// TIA Portal project "Servo With PLC" (V18)

(* hardware
DEVICE "S7-1200 station_1"  S7-1200 Station
   slot 0: "Rack_0"  S7-1200 Rack  Rack  V1.0
   slot 1: "PLC_1"  CPU 1215C DC/DC/DC  6ES7 215-1AG40-0XB0  V4.6
*)

// ===== PLC "PLC_1"  CPU 1215C DC/DC/DC =====

VAR_GLOBAL   // PLC tag table "Default tag table"
   "Servo Control_Pulse" AT %Q0.0 : Bool;
   "Servo Control_Direction" AT %Q0.1 : Bool;
   "Servo Control_DriveEnable" AT %Q0.2 : Bool;
   "Tag_1" AT %M0.0 : Bool;
   "Tag_2" AT %M0.1 : Bool;
   "Tag_3" AT %M0.2 : Bool;
   "Tag_4" AT %M0.3 : Bool;
   "Velocity for JOG" AT %MD10 : Real;
   "Tag_5" AT %M0.4 : Bool;
   "Tag_6" AT %MD14 : Real;
   "Tag_7" AT %MD18 : Real;
   "TotalTime (S)" AT %MD22 : Real;
   "tagg" AT %MD26 : Real;
   "Final Distance (mm)" AT %MD24 : Real;
   "final distance (mm)(1)" AT %MD30 : Real;
   "Tag_8" AT %M0.5 : Bool;
   "Tag_9" AT %M0.6 : Bool;
   "Tag_10" AT %MD34 : Real;
   "Tag_11" AT %MD38 : Real;
END_VAR

DATA_BLOCK "Servo Control"   // DB1, Motion_DB
{ S7_Optimized_Access := 'TRUE' }
AUTHOR : SIMATIC
FAMILY : BasicMC
NAME : TO_PosAx
VERSION : 8.0
// stored: InstanceOfName TO_PositioningAxis
"TO_PositioningAxis"
BEGIN
   // Axis.EnableOutput_AddressCU = %Q0.2
   // Axis.LengthUnit.LastDistance = -1
   // Axis.OnlinePtoModeCU = 16#0000_0002
   // Axis.DirectionOutputEnabledCU = TRUE
   // Axis.SelectedChannel2EnumCU = %Q0.1
   // Axis.SelectedChannel1EnumCU = %Q0.0
   // Pulse.MinDeltaDeltaFrequencyCU = 0.004
   // Pulse.MaxDeltaDeltaFrequencyCU = 1.0E+10
   // Pulse.MinDeltaFrequencyCU = 0.005
   // Pulse.MaxDeltaFrequencyCU = 9.5E+9
   // Pulse.MinFrequencyCU = 1.0
   // Pulse.MaxFrequencyCU = 100000.0
   // Pulse.OutputSourceCU = 16#0000_0000
   // Axis.SelectPTO = 0
END_DATA_BLOCK

ORGANIZATION_BLOCK "Main"   // OB1, LAD, ProgramCycle
TITLE = "Main Program Sweep (Cycle)"
{ S7_Optimized_Access := 'TRUE' }
VERSION : 0.1
   VAR_INPUT
      Initial_Call : Bool;   // Initial call of this OB
      Remanence : Bool;   // =True, if remanent data are available
   END_VAR
BEGIN

REGION Network 1
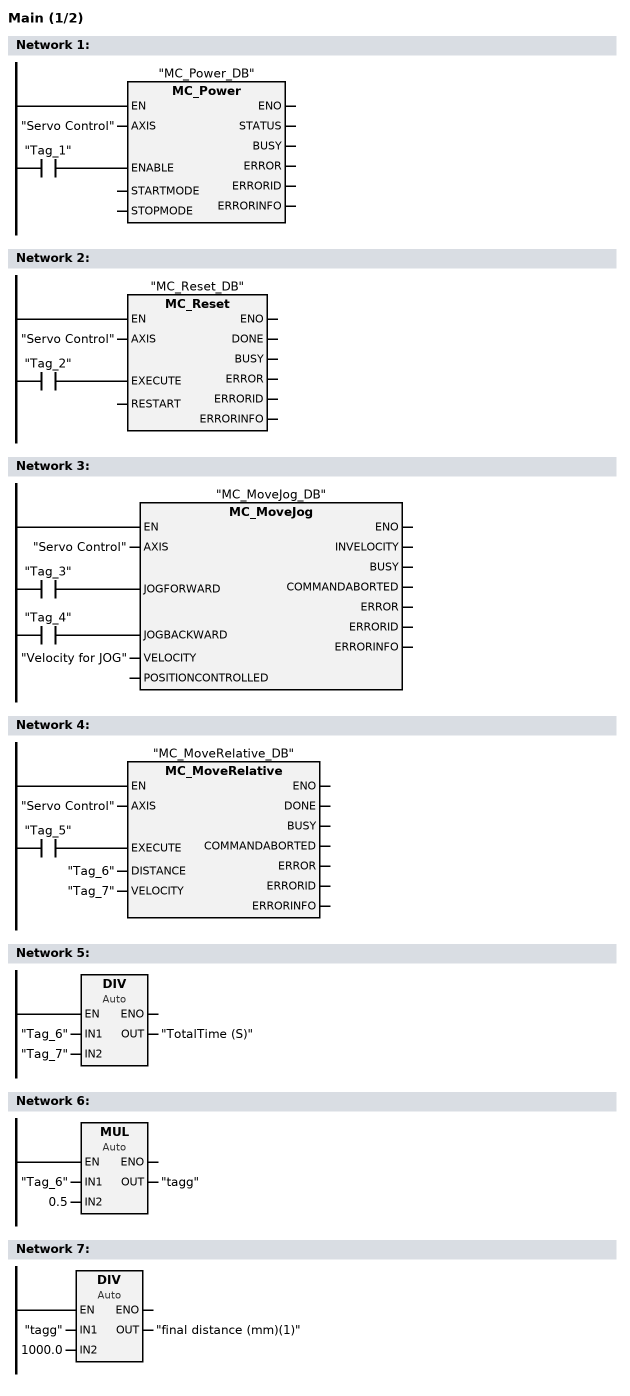
   "MC_Power_DB"(Axis := "Servo Control", Enable := "Tag_1");   // MC_Power
END_REGION

REGION Network 2
   "MC_Reset_DB"(Axis := "Servo Control", Execute := "Tag_2");   // MC_Reset
END_REGION

REGION Network 3
   "MC_MoveJog_DB"(Axis := "Servo Control",   // MC_MoveJog
                   JogForward := "Tag_3",
                   JogBackward := "Tag_4",
                   Velocity := "Velocity for JOG");
END_REGION

REGION Network 4
   "MC_MoveRelative_DB"(Axis := "Servo Control", Execute := "Tag_5", Distance := "Tag_6", Velocity := "Tag_7");   // MC_MoveRelative
END_REGION

REGION Network 5
   RUNG wire#powerrail
      Div(in1 := "Tag_6", in2 := "Tag_7", out => "TotalTime (S)")
   END_RUNG
   // the same network as SCL:
   "TotalTime (S)" := "Tag_6" / "Tag_7";
END_REGION

REGION Network 6
   RUNG wire#powerrail
      Mul(in1 := "Tag_6", in2 := 0.5, out => "tagg")
   END_RUNG
   // the same network as SCL:
   "tagg" := "Tag_6" * 0.5;
END_REGION

REGION Network 7
   RUNG wire#powerrail
      Div(in1 := "tagg", in2 := 1000.0, out => "final distance (mm)(1)")
   END_RUNG
   // the same network as SCL:
   "final distance (mm)(1)" := "tagg" / 1000.0;
END_REGION

REGION Network 8
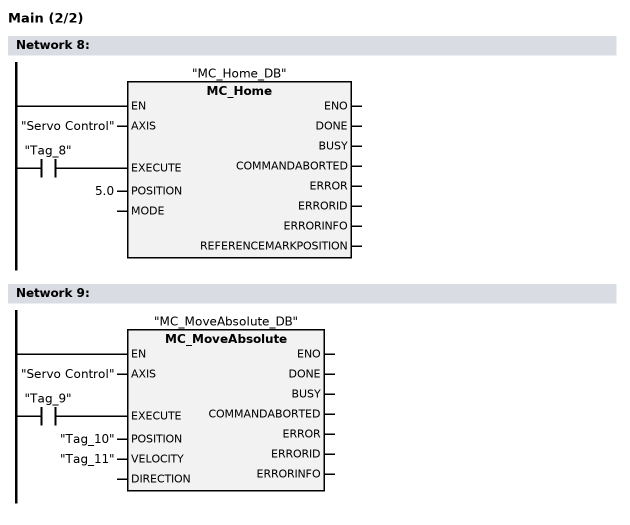
   "MC_Home_DB"(Axis := "Servo Control", Execute := "Tag_8", Position := 5.0);   // MC_Home
END_REGION

REGION Network 9
   "MC_MoveAbsolute_DB"(Axis := "Servo Control", Execute := "Tag_9", Position := "Tag_10", Velocity := "Tag_11");   // MC_MoveAbsolute
END_REGION
END_ORGANIZATION_BLOCK